VAR_GLOBAL
    {attribute 'pytmc' := 'pv: QRIX:SA:ESTOP_RST'}
    bResetIClk: BOOL;
    {attribute 'pytmc' := 'pv: QRIX:SA:ESTOP'}
    {attribute 'TcLinkTo' := 'TIIB[Rack#1A-02 SFIN (EL1918)]^StandardInputs^Standard Out Var 18'}
    bESTOP AT %I*: BOOL;

    {attribute 'TcLinkTo' := 'TIIB[Rack#2B-05 SV_AIR (EL2004)]^Channel 1^Output'}
    {attribute 'pytmc' := 'pv: QRIX:SA:SV1'}
    bOpenSV1 AT %Q*: BOOL;
    {attribute 'TcLinkTo' := 'TIIB[Rack#2B-05 SV_AIR (EL2004)]^Channel 2^Output'}
    {attribute 'pytmc' := 'pv: QRIX:SA:SV2'}
    bOpenSV2 AT %Q*: BOOL;

    {attribute 'TcLinkTo' := 'TIIB[Rack#1C_ServoDR (NCR-HD Series)]^260th receive PDO Mapping^Positive torque limit value'}
    iServoTorqueLimitPositive AT %Q*: UINT;

    {attribute 'TcLinkTo' := 'TIIB[Rack#1C_ServoDR (NCR-HD Series)]^260th receive PDO Mapping^Negative torque limit value'}
    iServoTorqueLimitNegative AT %Q*: UINT;

END_VAR

(* stored: Version 1.1.0.1, ProductVersion 3.1.4022.18
   GVL GVL_EPS: Id {d80bcb88-755c-4636-a81b-aa32affdb6ed} *)
